Staubli VAL3: stop.pgx

program stop()
begin
  homePointCopy = homePoint
  popUpMsg("Pending movement commands have been canceled")
  resetMotion()
end
